{attribute 'qualified_only'}
{attribute 'strict'}
TYPE eSensorError :
(
	CommunicationError := 0,	
	OutOfRange := 1,
	UndefinedError := 2,
	NoError	:= 3
);
END_TYPE

(* stored: Version 1.1.0.1, ProductVersion 3.1.4024.12
   DUT eSensorError: Id {3a850c02-3d91-4e9f-94d7-922f70e1c714} *)
